(* LS Electric XG5000 project: 20230517_PLC_Function_Block *)
(* PLC LSPLC *)

PROGRAM NewProgram (* task: 스캔 프로그램 *)
VAR
    LAG : TON;
    on : BOOL;
    OPEN : TON;
    RESET : TON;
    T1 : TON;
    T1_스위치 : BOOL;
    T2 : TOF;
    T2_스위치 : BOOL;
    T3 : TP;
    T3_스위치 : BOOL;
    T4 : TON;
    T4_스위치 : BOOL;
    T5 : TON;
    T6 : TON;
    T6_스위치 : BOOL;
    T7 : TON;
    T7_스위치 : BOOL;
    T8 : TON;
    T9 : TON;
    T9_OFF : TOF;
    time02 : TIME;
    time03 : TIME;
    timer1 : TON;
    timer2 : TP;
    timer3 : TP;
    timer4 : TON;
    timer5 : TOF;
    timer6 : TP;
    TON_INST : TON;
    깜빡 : BOOL;
    램프1 : BOOL;
    램프2 : BOOL;
    램프3 : BOOL;
    램프4 : BOOL;
    램프5 : BOOL;
    물 : BOOL;
    변기 : BOOL;
    비데 : BOOL;
    비데2 : BOOL;
    센서 : BOOL;
    센서2 : BOOL;
    입력 : BOOL;
    정지 : BOOL;
    조명 : BOOL;
END_VAR
VAR
    _e1 : R_TRIG;
    _e2 : R_TRIG;
END_VAR

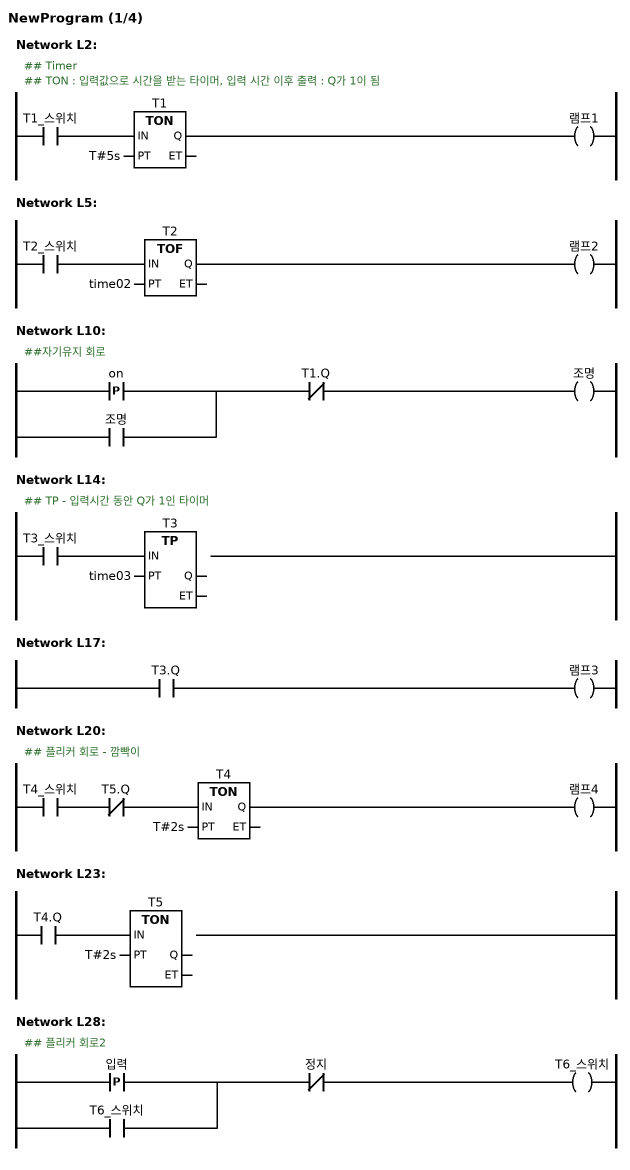
(* ## Timer *)
(* ## TON : 입력값으로 시간을 받는 타이머, 입력 시간 이후 출력 : Q가 1이 됨 *)
(* Rung L2 *)
T1(IN := T1_스위치, PT := T#5s);
램프1 := T1.Q;
(* Rung L5 *)
T2(IN := T2_스위치, PT := time02);
램프2 := T2.Q;
(* ##자기유지 회로 *)
(* Rung L10 *)
_e1(CLK := on);
조명 := (_e1.Q OR 조명) AND NOT T1.Q;
(* ## TP - 입력시간 동안 Q가 1인 타이머 *)
(* Rung L14 *)
T3(IN := T3_스위치, PT := time03);
(* Rung L17 *)
램프3 := T3.Q;
(* ## 플리커 회로 - 깜빡이 *)
(* Rung L20 *)
T4(IN := T4_스위치 AND NOT T5.Q, PT := T#2s);
램프4 := T4.Q;
(* Rung L23 *)
T5(IN := T4.Q, PT := T#2s);
(* ## 플리커 회로2 *)
(* Rung L28 *)
_e2(CLK := 입력);
T6_스위치 := (_e2.Q OR T6_스위치) AND NOT 정지;

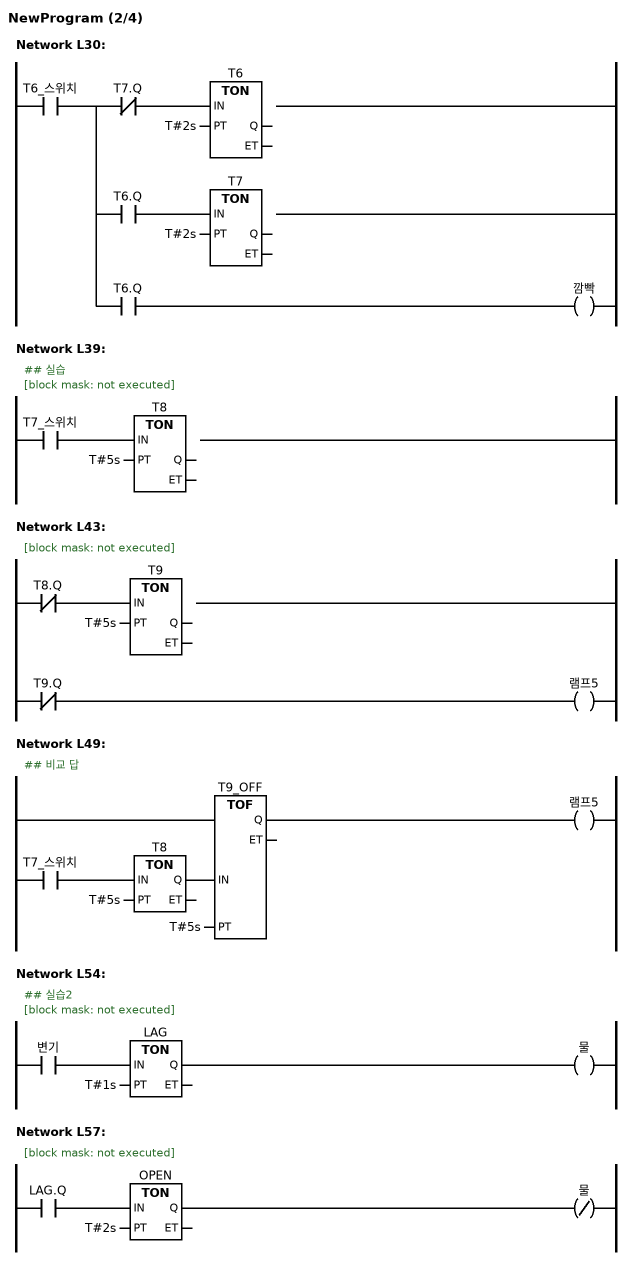
(* Rung L30 *)
T6(IN := T6_스위치 AND NOT T7.Q, PT := T#2s);
T7(IN := T6_스위치 AND T6.Q, PT := T#2s);
깜빡 := T6_스위치 AND T6.Q;
(* ## 실습 *)
(* Rung L39 is block-masked: not executed *)
// T8(IN := T7_스위치, PT := T#5s);
(* Rung L43 is block-masked: not executed *)
// T9(IN := NOT T8.Q, PT := T#5s);
// 램프5 := NOT T9.Q;
(* ## 비교 답 *)
(* Rung L49 *)
T8(IN := T7_스위치, PT := T#5s);
T9_OFF(IN := T8.Q, PT := T#5s);
램프5 := T9_OFF.Q;
(* ## 실습2 *)
(* Rung L54 is block-masked: not executed *)
// LAG(IN := 변기, PT := T#1s);
// 물 := LAG.Q;
(* Rung L57 is block-masked: not executed *)
// OPEN(IN := LAG.Q, PT := T#2s);
// 물 := NOT OPEN.Q;

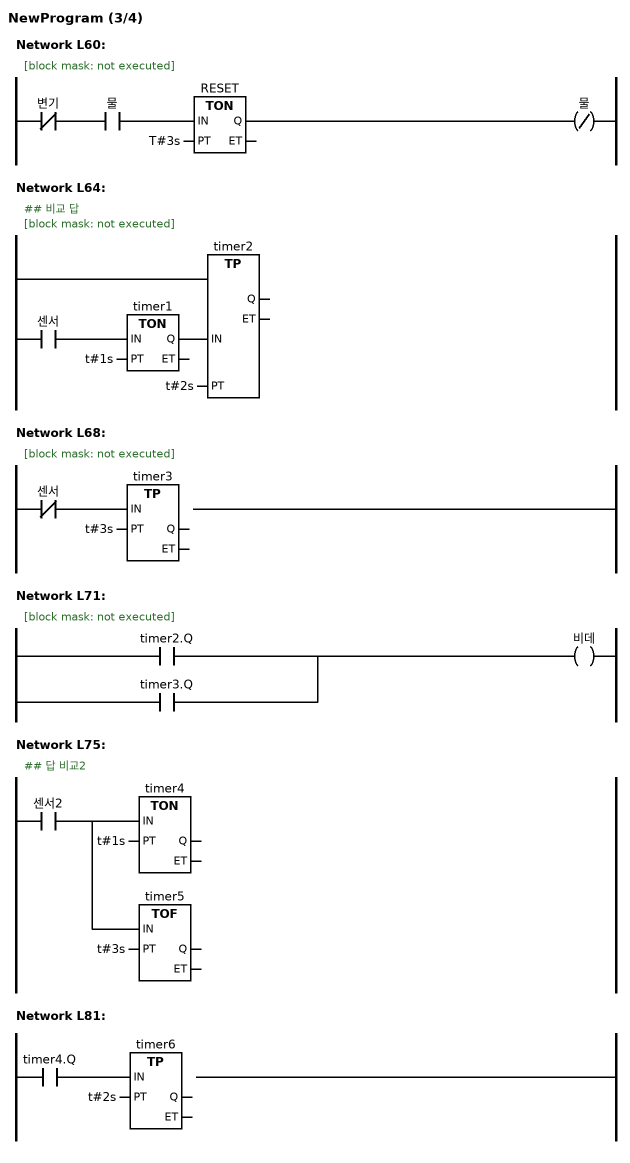
(* Rung L60 is block-masked: not executed *)
// RESET(IN := NOT 변기 AND 물, PT := T#3s);
// 물 := NOT RESET.Q;
(* ## 비교 답 *)
(* Rung L64 is block-masked: not executed *)
// timer1(IN := 센서, PT := t#1s);
// timer2(IN := timer1.Q, PT := t#2s);
(* Rung L68 is block-masked: not executed *)
// timer3(IN := NOT 센서, PT := t#3s);
(* Rung L71 is block-masked: not executed *)
// 비데 := timer2.Q OR timer3.Q;
(* ## 답 비교2 *)
(* Rung L75 *)
timer4(IN := 센서2, PT := t#1s);
timer5(IN := 센서2, PT := t#3s);
(* Rung L81 *)
timer6(IN := timer4.Q, PT := t#2s);

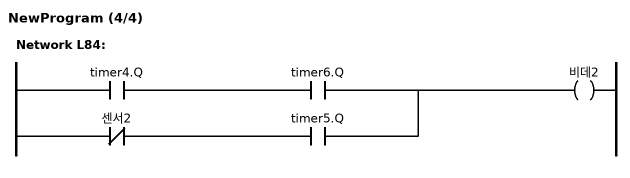
(* Rung L84 *)
비데2 := (timer4.Q AND timer6.Q) OR (NOT 센서2 AND timer5.Q);
END_PROGRAM